// TIA Portal V19 export
TYPE "UDT_DIFF"
   STRUCT
      sim : Struct   // Simulation
         en { S7_SetPoint := 'True'} : Bool := false;   // Simulation command
         value { S7_SetPoint := 'True'} : Real := 0.0;   // Simulation value
      END_STRUCT;
      faults : Struct   // Alarms
         hh { S7_SetPoint := 'True'} : "UDT_ALARMACKN";   // UDT_DELAYONOFF
         h { S7_SetPoint := 'True'} : "UDT_ALARMACKN";   // UDT_DELAYONOFF
         l { S7_SetPoint := 'True'} : "UDT_ALARMACKN";   // UDT_DELAYONOFF
         ll { S7_SetPoint := 'True'} : "UDT_ALARMACKN";   // UDT_DELAYONOFF
         sp_hh { S7_SetPoint := 'True'} : Real := 0.0;   // Setpoint of high-high alarm
         sp_h { S7_SetPoint := 'True'} : Real := 0.0;   // Setpoint of high alarm
         sp_l { S7_SetPoint := 'True'} : Real := 0.0;   // Setpoint of low alarm
         sp_ll { S7_SetPoint := 'True'} : Real := 0.0;   // Setpoint of low-low alarm
         fpreset : Bool := false;   // Reset Alarms
      END_STRUCT;
      minuend : Real := 0.0;   // Minuend
      subtrahend : Real := 0.0;   // Subtrahend
      trendhigh { S7_SetPoint := 'True'} : Real := 0.0;   // 120% High limit of scale process. Used for trend axis
      output : Real := 0.0;   // Differential output
      unit : WString := WSTRING#'';
   END_STRUCT;
END_TYPE
